// TIA Portal V17 export
// export: Created 2024-09-03T21:55:01.5642694Z, ExportSetting WithDefaults, DisplayName Totally Integrated Automation Portal, DisplayVersion V17 Update 7, DisplayName TIA Portal Openness, DisplayVersion V17 Update 7, DisplayName TIA Portal Version Control Interface, DisplayVersion V17, DisplayName SINAMICS Startdrive Advanced, DisplayVersion V17 SP2, DisplayName SINAMICS Startdrive G110M, G120, G120C, G120D, G120P, G115D, DisplayVersion V17 SP2, DisplayName SINAMICS Startdrive G130, G150, S120, S150, SINAMICS MV, S210, DisplayVersion V17 SP2, DisplayName STEP 7 Professional, DisplayVersion V17 Update 7, DisplayName STEP 7 Safety, DisplayVersion V17 Update 6, DisplayName WinCC Advanced / Unified PC, DisplayVersion V17 Update 7
DATA_BLOCK "DB_STATUS_IJCORE"   // DB69
{ S7_Optimized_Access := 'TRUE' }
VERSION : 0.1
// stored: AutoNumber true, DBAccessibleFromOPCUA true, DBAccessibleFromWebserver true, IsOnlyStoredInLoadMemory false, IsRetainMemResEnabled false, IsWriteProtectedInAS false, MemoryReserve 100
   VAR
      CONFIG_MSG { S7_SetPoint := 'True'} : Array[0..30] of "CONFIG_MSG_IJC";
      EDIT_MSG { S7_SetPoint := 'True'} : "CONFIG_MSG_IJC";
      INDEX_EDITADO { S7_SetPoint := 'True'} : Int := 1;
      INDEX_EDITADO_ANTERIOR : Int := 1;
      PB_VALIDAR_EDICION { S7_SetPoint := 'True'} : Bool := FALSE;
      ANSWER_RECIB : Array[0..30] of Int;
      ANSWER_NFP : Array[0..5] of Int;
      ANSWER_TRB : Array[0..5] of Int;
      ANSWER_STA : Array[0..5] of Int;
      ANSWER_TRC : Array[0..5] of Int;
      ANSWER_TRW : Array[0..5] of Int;
      ANSWER_TRI : Array[0..5] of Int;
      DN_TRC_COMP : Array[0..5] of Bool;
      ALL_TRC_OK : Bool;
      ALL_CNF_OK : Bool;
      ALL_TRR_OK : Bool;
      INDEX_ENVIO : DInt := 40;
      INDEX_MSG_CONFIG : DInt;
      ALARMA : Array[0..10] of Word;
      INDEX_ANSWER_STA : Int := 0;
      INDEX_ANSWER_TRC : Int := 9;
      INDEX_ANSWER_TRW : Int := 15;
      INDEX_ANSWER_TRI : Int := 10;
      INDEX_CLEAR : Int;
      INDEX_HMI : Int;
      PAGINA_HMI : Int;
      PAGINA_UP : Bool;
      PAGINA_DOWN : Bool;
      HMI_M_TYPE : Array[0..10] of String;
      HMI_M_NBR : Array[0..10] of DInt;
      HMI_ANS : Array[0..10] of SInt;
      HMI_STEP : Array[0..10] of Int;
      HMI_FLT : Array[0..10] of Bool;
      HMI_DN : Array[0..10] of Bool;
      HMI : Array[0..10] of Struct
         SEND : Struct
            MSG : String[50];
            SW : SInt;
         END_STRUCT;
         RCV : Struct
            MSG : String[50];
            SW : SInt;
         END_STRUCT;
      END_STRUCT;
      AW_number : DInt;
      AW_duration : Time;
      AW_durationMax : Time;
      Restart_Counter_bit_of_life : Int;
      AW_duration_fault : Time;
      R_NBR_MESSAGE : DInt;
      MES_DIAG_MESSAGE_NBR : Int := 1;
      S_DURATION_FAULT : Int := 30;
      R_DURATION_FAULT : Int := 30;
      S_DURATION : Int;
      S_MAX_DURATION : Int;
      S_NBR_MESSAGE : DInt;
      R_DURATION : Int;
      R_MAX_DURATION : Int;
      MES_RESET_AW_DIAG : Bool;
      MES_RESET_MESS_DIAG : Bool;
      MES_TEMP_S_FT : Int := 30;
      MES_TEMP_R_FT : Int := 30;
      MES_TEMP_NBR_MESS : Int := 1;
   END_VAR
BEGIN
   CONFIG_MSG[1..4]."TYPE" := 'STA';
   CONFIG_MSG[5..8]."TYPE" := 'TRC';
   CONFIG_MSG[9..10]."TYPE" := 'TRR';
   CONFIG_MSG[11..14]."TYPE" := 'CNF';
   CONFIG_MSG[15]."TYPE" := 'PFC';
   EDIT_MSG."TYPE" := '';
   EDIT_MSG.KANBAN := '';
   EDIT_MSG.COMPONENT := '';
   EDIT_MSG.START := FALSE;
   EDIT_MSG.PROCESS_STATUS := 0;
   ANSWER_RECIB[0..2] := 0;
   ANSWER_RECIB[3] := 1;
   ANSWER_RECIB[4..5] := 8224;
   ANSWER_RECIB[6] := 1;
   ANSWER_RECIB[7..8] := 8224;
   ANSWER_RECIB[9..11] := 0;
   ANSWER_RECIB[12] := 1;
   ANSWER_RECIB[13..14] := 8224;
   ANSWER_RECIB[15..18] := 0;
   ANSWER_RECIB[19] := 1;
   ANSWER_RECIB[20] := 8224;
   ANSWER_NFP[0..2] := 0;
   ANSWER_NFP[3] := 1;
   ANSWER_NFP[4..5] := 8224;
   ANSWER_TRB[0..5] := 0;
   ANSWER_STA[0..2] := 0;
   ANSWER_STA[3..4] := 1;
   ANSWER_STA[5] := 0;
   ANSWER_TRC[0..5] := 0;
   ANSWER_TRW[0..5] := 0;
   ANSWER_TRI[0..5] := 0;
   DN_TRC_COMP[0..5] := FALSE;
   ALARMA[0..10] := 16#0000;
END_DATA_BLOCK
